Fanuc KAREL source: V_GET_FOUND.kl

PROGRAM T
%NOLOCKGROUP
VAR
 v0 : STRING[40]
 v1 : INTEGER
 v2 : INTEGER
 v3 : INTEGER
 v4 : XYZWPR
 v5 : ARRAY[5] OF XYZWPR
 v6 : ARRAY[10] OF REAL
 v7 : INTEGER
BEGIN
 V_GET_FOUND(v0, v1, v2, v3, v4, v5, v6, v7)
END T
